// S11 rig instance. Test image only, like the S2 harness.
DATA_BLOCK "S11Rig"
{ S7_Optimized_Access := 'TRUE' }
VERSION : 0.1
NON_RETAIN
"FB_SpkGraphRig"

BEGIN

END_DATA_BLOCK
